DATA_BLOCK "ST10_Flow11_A2TableScan_iDB"
{ S7_Optimized_Access := 'TRUE' }
VERSION : 0.1
NON_RETAIN
"ST10_Flow11_A2TableScan"

BEGIN

END_DATA_BLOCK

